// TIA Portal V20 export
DATA_BLOCK "Config"   // DB169
// stored: MemoryReserve 100, Namespace Unit1.Em2
   VAR
      em : "LAF_typeEmConfiguration";   // Configuration of EM Parameters
   END_VAR
   VAR RETAIN
      cmElectrodeFixRightTopFwdBwd : "LBC_typeTwoWayActuatorConfiguration";
      cmElectrodeFixRightBottomFwdBwd : "LBC_typeTwoWayActuatorConfiguration";
      cmElectrodeFixLeftTopFwdBwd : "LBC_typeTwoWayActuatorConfiguration";
      cmElectrodeFixLeftBottomFwdBwd : "LBC_typeTwoWayActuatorConfiguration";
      cmElectrodeFixLeftTopUpDown : "LBC_typeTwoWayActuatorConfiguration";
      cmElectrodeFixLeftBottomUpDown : "LBC_typeTwoWayActuatorConfiguration";
      cmUwSemiSplicerVacuumRightTopOnOff : "LBC_typeTwoWayActuatorConfiguration";
      cmUwSemiSplicerVacuumRightBottomOnOff : "LBC_typeTwoWayActuatorConfiguration";
      cmUwSemiSplicerVacuumLeftTopOnOff : "LBC_typeTwoWayActuatorConfiguration";
      cmUwSemiSplicerVacuumLeftBottomOnOff : "LBC_typeTwoWayActuatorConfiguration";
      cmElectrodeCutterFwdBwd : "LBC_typeTwoWayActuatorConfiguration";
      cmSplicingLeftModuleMoverFwdBwd : "LBC_typeTwoWayActuatorConfiguration";
      cmSplicingRightModuleMoverFwdBwd : "LBC_typeTwoWayActuatorConfiguration";
      cmElectrodeLeftHolderMoverFwdBwd : "LBC_typeTwoWayActuatorConfiguration";
      cmElectrodeRightHolderMoverFwdBwd : "LBC_typeTwoWayActuatorConfiguration";
      cmTapeLoadingTurnCwCcw : "LBC_typeTwoWayActuatorConfiguration";
      cmTapeAttachUnitFwdBwd : "LBC_typeTwoWayActuatorConfiguration";
      cmTapeVacuumOnOff : "LBC_typeTwoWayActuatorConfiguration";
      cmStopperFwdBwd : "LBC_typeTwoWayActuatorConfiguration";
      cmSupportUnitTransferFwdBwd : "LBC_typeTwoWayActuatorConfiguration";
      cmSupportUnitShaftUpDown : "LBC_typeTwoWayActuatorConfiguration";
      cmFrameCoverFwdBwd : "LBC_typeTwoWayActuatorConfiguration";
      TapeAttachRetryCountSV : Int;
   END_VAR
BEGIN
   cmTapeLoadingTurnCwCcw.monitoringDiscrepancy := T#1s;
END_DATA_BLOCK
